// Brief: Master Arm Initialization
FUNCTION_BLOCK PUBLIC FB_ArmError EXTENDS FB_MasterArmCtrlBase
VAR_INPUT
END_VAR
VAR_OUTPUT
END_VAR
VAR
END_VAR

END_FUNCTION_BLOCK

(* stored: Version 1.1.0.1, ProductVersion 3.1.4024.12
   POU FB_ArmError: Id {78b2e60d-537e-446e-8b3b-6db63d5ab02c}, SpecialFunc None *)
